// TIA Portal V16 export
// export: Created 2022-07-21T09:35:23.8288395Z, ExportSetting WithDefaults, DisplayName Totally Integrated Automation Portal, DisplayVersion V16 Update 4, DisplayName TIA Portal Version Control Interface, DisplayVersion V16 Update 2, DisplayName TIA Portal Openness, DisplayVersion V16 Update 4, DisplayName SINAMICS Startdrive Advanced, DisplayVersion V16 Update 5, DisplayName SINAMICS Startdrive G130, G150, S120, S150, SINAMICS MV, S210, DisplayVersion V16 Update 5, DisplayName SINAMICS Startdrive G110M, G120, G120C, G120D, G120P, G115D, DisplayVersion V16 Update 5, DisplayName STEP 7 Professional, DisplayVersion V16 Update 4, DisplayName STEP 7 Safety, DisplayVersion V16, DisplayName WinCC Advanced, DisplayVersion V16 Update 4
FUNCTION "fcFeedFunctionButtons" : Void   // FC13, LAD
TITLE = Special function buttons / Przyciski funkcji specjalnych
{ S7_Optimized_Access := 'TRUE' }
VERSION : 0.1
// stored: AutoNumber false, IsIECCheckEnabled false, SetENOAutomatically false, UDAEnableTagReadback false
   VAR_IN_OUT
      io : "typeInterrollCtrl";
   END_VAR
BEGIN

REGION Network 1: Trigger acknowledge window / Wyzwolenie okna potwierdzenia
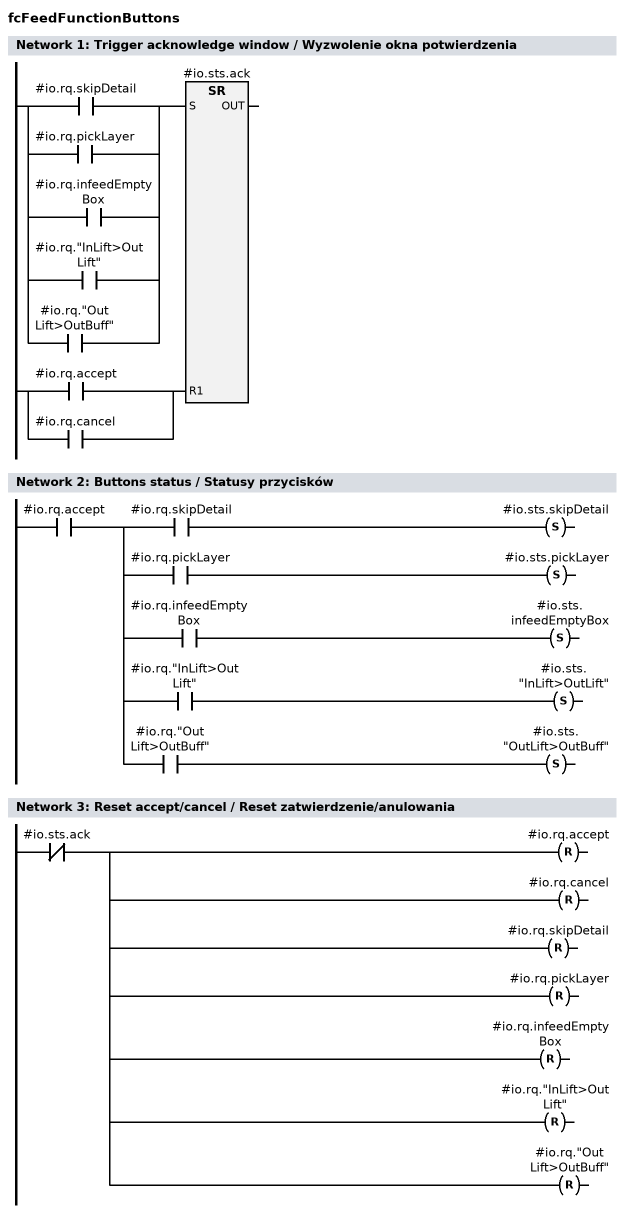
   RUNG wire#powerrail
      Contact( #io.rq.skipDetail )
      wire#w1
      S_SR(operand := #io.sts.ack, r1 := wire#w2)
   END_RUNG
   RUNG wire#powerrail
      Contact( #io.rq.pickLayer )
   END_RUNG wire#w1
   RUNG wire#powerrail
      Contact( #io.rq.infeedEmptyBox )
   END_RUNG wire#w1
   RUNG wire#powerrail
      Contact( #io.rq."InLift>OutLift" )
   END_RUNG wire#w1
   RUNG wire#powerrail
      Contact( #io.rq."OutLift>OutBuff" )
   END_RUNG wire#w1
   RUNG wire#powerrail
      Contact( #io.rq.accept )
   END_RUNG wire#w2
   RUNG wire#powerrail
      Contact( #io.rq.cancel )
   END_RUNG wire#w2
   // the same network as SCL:
   IF #io.rq.skipDetail OR #io.rq.pickLayer OR #io.rq.infeedEmptyBox OR #io.rq."InLift>OutLift" OR #io.rq."OutLift>OutBuff" THEN
       #io.sts.ack := TRUE;   // SR flip-flop
   END_IF;
   IF #io.rq.accept OR #io.rq.cancel THEN #io.sts.ack := FALSE; END_IF;
END_REGION

REGION Network 2: Buttons status / Statusy przycisków
   RUNG wire#powerrail
      Contact( #io.rq.accept )
      wire#w1
      Contact( #io.rq.skipDetail )
      S_Coil( #io.sts.skipDetail )
   END_RUNG
   RUNG wire#w1
      Contact( #io.rq.pickLayer )
      S_Coil( #io.sts.pickLayer )
   END_RUNG
   RUNG wire#w1
      Contact( #io.rq.infeedEmptyBox )
      S_Coil( #io.sts.infeedEmptyBox )
   END_RUNG
   RUNG wire#w1
      Contact( #io.rq."InLift>OutLift" )
      S_Coil( #io.sts."InLift>OutLift" )
   END_RUNG
   RUNG wire#w1
      Contact( #io.rq."OutLift>OutBuff" )
      S_Coil( #io.sts."OutLift>OutBuff" )
   END_RUNG
   // the same network as SCL:
   IF #io.rq.accept AND #io.rq.skipDetail THEN #io.sts.skipDetail := TRUE; END_IF;
   IF #io.rq.accept AND #io.rq.pickLayer THEN #io.sts.pickLayer := TRUE; END_IF;
   IF #io.rq.accept AND #io.rq.infeedEmptyBox THEN #io.sts.infeedEmptyBox := TRUE; END_IF;
   IF #io.rq.accept AND #io.rq."InLift>OutLift" THEN #io.sts."InLift>OutLift" := TRUE; END_IF;
   IF #io.rq.accept AND #io.rq."OutLift>OutBuff" THEN #io.sts."OutLift>OutBuff" := TRUE; END_IF;
END_REGION

REGION Network 3: Reset accept/cancel / Reset zatwierdzenie/anulowania
   RUNG wire#powerrail
      I_Contact( #io.sts.ack )
      wire#w1
      R_Coil( #io.rq.accept )
   END_RUNG
   RUNG wire#w1
      R_Coil( #io.rq.cancel )
   END_RUNG
   RUNG wire#w1
      R_Coil( #io.rq.skipDetail )
   END_RUNG
   RUNG wire#w1
      R_Coil( #io.rq.pickLayer )
   END_RUNG
   RUNG wire#w1
      R_Coil( #io.rq.infeedEmptyBox )
   END_RUNG
   RUNG wire#w1
      R_Coil( #io.rq."InLift>OutLift" )
   END_RUNG
   RUNG wire#w1
      R_Coil( #io.rq."OutLift>OutBuff" )
   END_RUNG
   // the same network as SCL:
   IF NOT #io.sts.ack THEN
       #io.rq.accept := FALSE;
       #io.rq.cancel := FALSE;
       #io.rq.skipDetail := FALSE;
       #io.rq.pickLayer := FALSE;
       #io.rq.infeedEmptyBox := FALSE;
       #io.rq."InLift>OutLift" := FALSE;
       #io.rq."OutLift>OutBuff" := FALSE;
   END_IF;
END_REGION
END_FUNCTION
